(* PLC project CoDeSys External Library Template, WAGO e!COCKPIT e!COCKPIT, author 3S - Smart Software Solutions GmbH *)
(* stored: creationDateTime 2019-10-29T12:37:19.8256748, version 3.5.5.30, modificationDateTime 2019-10-29T12:36:39.3744516, organization 3S - Smart Software Solutions GmbH *)
(* Library project template with all possible element types, docu and a sample project structure *)

FUNCTION fnKomunikatDaneDoRaportu_REAL : STRING
  VAR_INPUT
    rWartosc : REAL;
    sAtrybut : STRING;
  END_VAR
  VAR_IN_OUT
    rWartoscZaraportowana : REAL;
    sDane : alSTRINGKomunikat;
  END_VAR

            IF rWartosc <> rWartoscZaraportowana THEN
	rWartoscZaraportowana := rWartosc;
	fnKomunikatDaneDodaj(sDane := sDane , sAtrybut := sAtrybut , sWartosc := REAL_TO_STRING(rWartosc));	
END_IF


          
END_FUNCTION
